// SIMATIC S7-200 project (STEP 7-Micro/WIN), CPU 224XP REL 02.01

SYMBOL_TABLE USUARIO1
P_MARCHA         I0.0
P_PARO           I0.1
TERMICO          I0.2
M1_LINEA         Q0.0
LED_MARCHA       Q0.1
M1_ESTRELLA      Q0.2
M1_TRIANGULO     Q0.3
LED_PARO         Q0.4
LED_AVERIA       Q0.5
END_SYMBOL_TABLE

SYMBOL_TABLE Símbolos S7-200
Primer_ciclo_ON  SM0.1    // ON sólo en el primer ciclo
END_SYMBOL_TABLE

ORGANIZATION_BLOCK PRINCIPAL:OB1
TITLE=COMENTARIOS DEL PROGRAMA
BEGIN
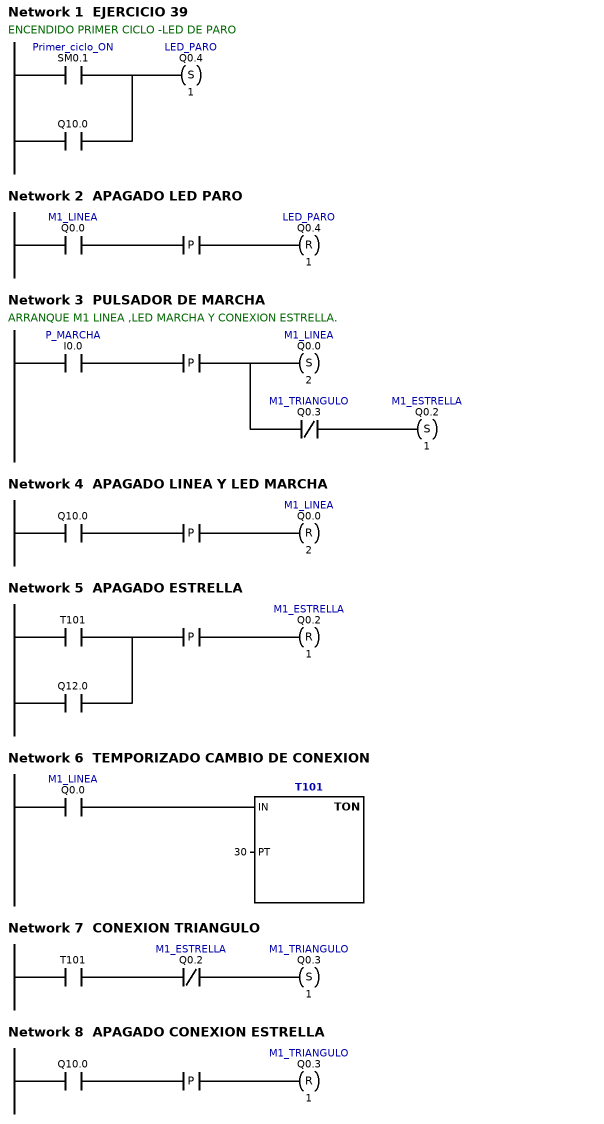
Network 1 // EJERCICIO 39
// ENCENDIDO PRIMER CICLO -LED DE PARO
LD     Primer_ciclo_ON:SM0.1
O      Q10.0
S      LED_PARO:Q0.4, 1
Network 2 // APAGADO LED PARO
LD     M1_LINEA:Q0.0
EU
R      LED_PARO:Q0.4, 1
Network 3 // PULSADOR DE MARCHA                            
// ARRANQUE M1 LINEA ,LED MARCHA Y CONEXION ESTRELLA.
LD     P_MARCHA:I0.0
EU
S      M1_LINEA:Q0.0, 2
AN     M1_TRIANGULO:Q0.3
S      M1_ESTRELLA:Q0.2, 1
Network 4 // APAGADO LINEA Y LED MARCHA
LD     Q10.0
EU
R      M1_LINEA:Q0.0, 2
Network 5 // APAGADO ESTRELLA
LD     T101
O      Q12.0
EU
R      M1_ESTRELLA:Q0.2, 1
Network 6 // TEMPORIZADO CAMBIO DE CONEXION
LD     M1_LINEA:Q0.0
TON    T101, 30
Network 7 // CONEXION TRIANGULO
LD     T101
AN     M1_ESTRELLA:Q0.2
S      M1_TRIANGULO:Q0.3, 1
Network 8 // APAGADO CONEXION ESTRELLA
LD     Q10.0
EU
R      M1_TRIANGULO:Q0.3, 1
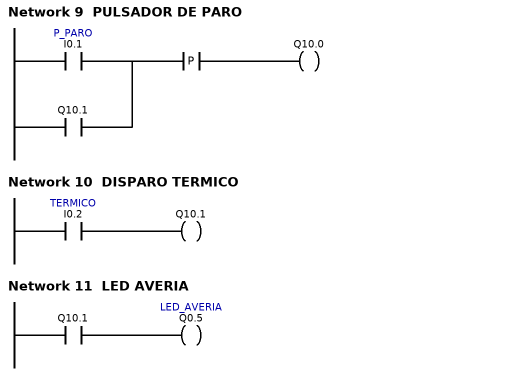
Network 9 // PULSADOR DE PARO
LD     P_PARO:I0.1
O      Q10.1
EU
=      Q10.0
Network 10 // DISPARO TERMICO
LD     TERMICO:I0.2
=      Q10.1
Network 11 // LED AVERIA
LD     Q10.1
=      LED_AVERIA:Q0.5
END_ORGANIZATION_BLOCK
